// Mitsubishi GX Works2 project: MPS 장비 제어 3   PLC: Q03UDV

PROGRAM MAIN
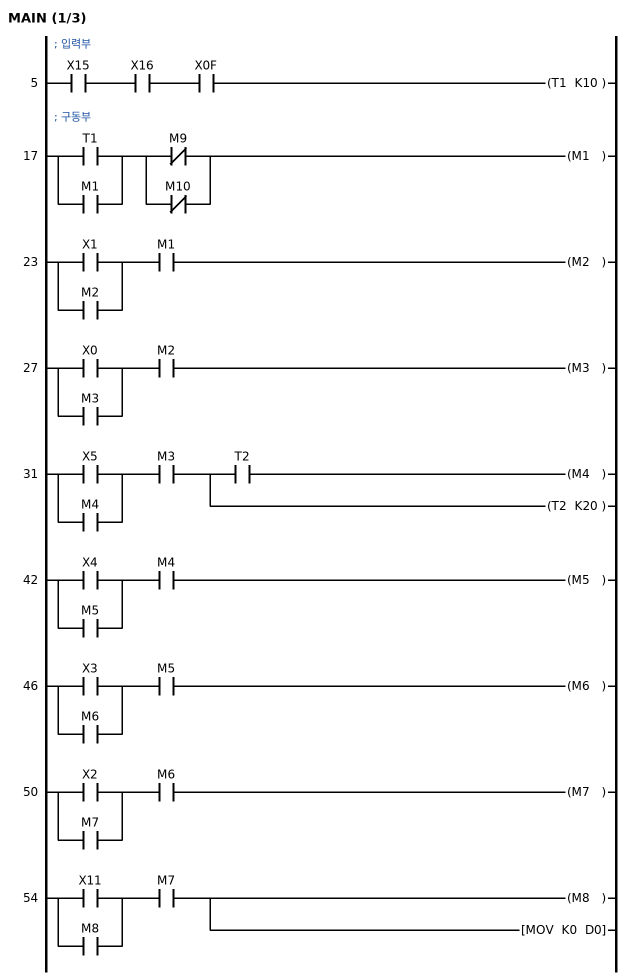
; 입력부
5     LD      X15
      AND     X16
      AND     X0F
      OUT     T1 K10
; 구동부
17    LD      T1
      OR      M1
      LDI     M9
      ORI     M10
      ANB
      OUT     M1
23    LD      X1
      OR      M2
      AND     M1
      OUT     M2
27    LD      X0
      OR      M3
      AND     M2
      OUT     M3
31    LD      X5
      OR      M4
      AND     M3
      MPS
      AND     T2
      OUT     M4
      MPP
      OUT     T2 K20
42    LD      X4
      OR      M5
      AND     M4
      OUT     M5
46    LD      X3
      OR      M6
      AND     M5
      OUT     M6
50    LD      X2
      OR      M7
      AND     M6
      OUT     M7
54    LD      X11
      OR      M8
      AND     M7
      OUT     M8
      MOV     K0 D0
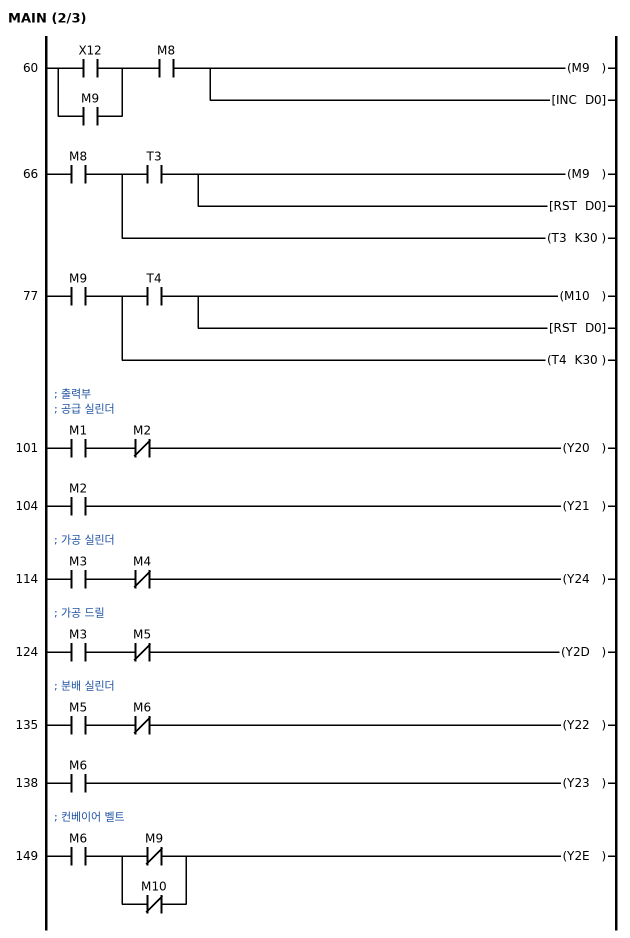
60    LD      X12
      OR      M9
      AND     M8
      OUT     M9
      INC     D0
66    LD      M8
      MPS
      AND     T3
      OUT     M9
      RST     D0
      MPP
      OUT     T3 K30
77    LD      M9
      MPS
      AND     T4
      OUT     M10
      RST     D0
      MPP
      OUT     T4 K30
; 출력부
; 공급 실린더
101   LD      M1
      ANI     M2
      OUT     Y20
104   LD      M2
      OUT     Y21
; 가공 실린더
114   LD      M3
      ANI     M4
      OUT     Y24
; 가공 드릴
124   LD      M3
      ANI     M5
      OUT     Y2D
; 분배 실린더
135   LD      M5
      ANI     M6
      OUT     Y22
138   LD      M6
      OUT     Y23
; 컨베이어 벨트
149   LD      M6
      LDI     M9
      ORI     M10
      ANB
      OUT     Y2E
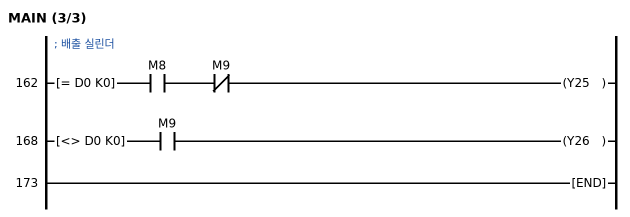
; 배출 실린더
162   LD=     D0 K0
      AND     M8
      ANI     M9
      OUT     Y25
168   LD<>    D0 K0
      AND     M9
      OUT     Y26
173   END
END_PROGRAM
